% RSLogix 500 project I2P JOB 12 - ANDREW_HOEMMEN_BAK049.RSS, saved by version 10.00.00.00 %
PROJECT "ML03A"    % processor: Bul.1763 MicroLogix 1100 Series B %

PROGRAM FILES
  LAD 2   8 rungs

DATA FILES
  O0 OUTPUT  4 elements
  I1 INPUT  6 elements
  S2 STATUS  66 elements
  B3 BINARY  1 elements
  T4 TIMER  1 elements
  C5 COUNTER  1 elements
  R6 CONTROL  1 elements
  N7 INTEGER  1 elements
  F8 FLOAT  1 elements

LADDER 2
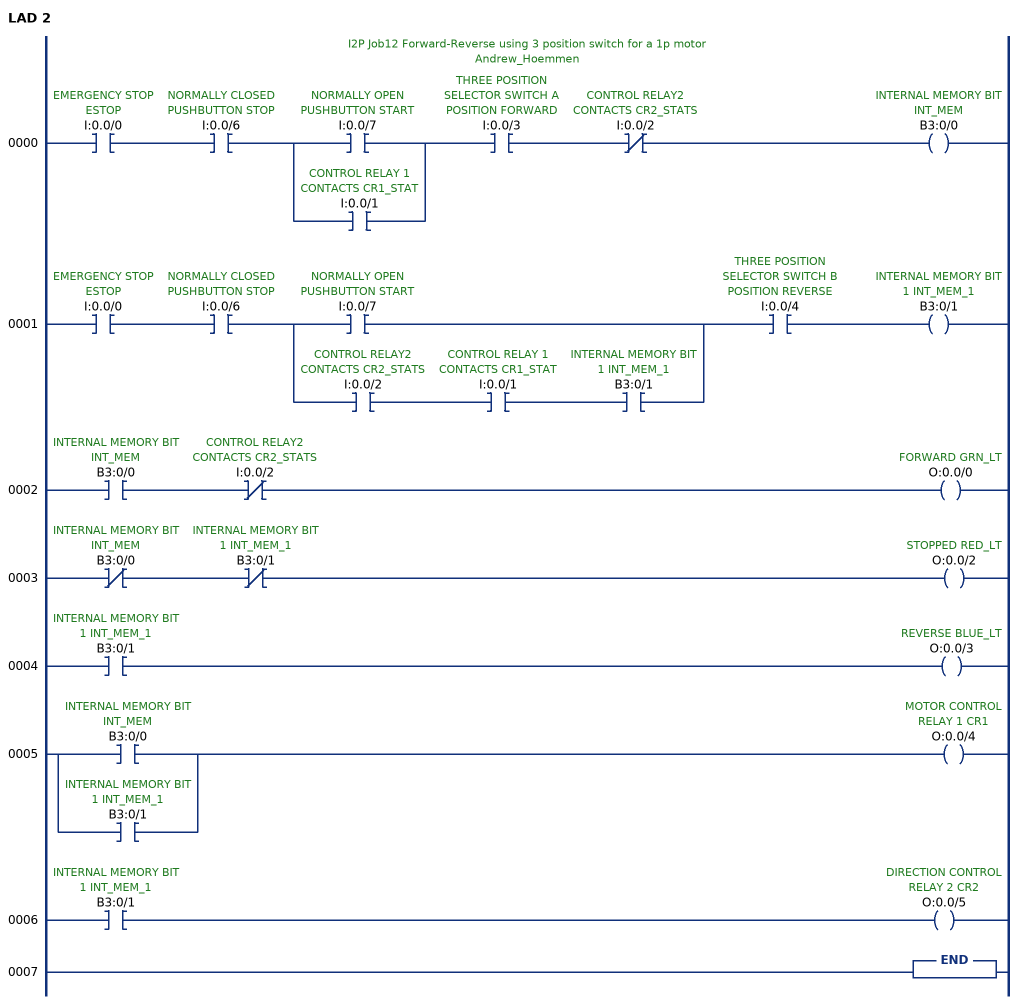
% Rung: 0 %
% I2P Job12 Forward-Reverse using 3 position switch for a 1p motor
% Andrew_Hoemmen %
SOR XIC I:0.0/0 XIC I:0.0/6 BST XIC I:0.0/7 NXB XIC I:0.0/1 BND XIC I:0.0/3 XIO I:0.0/2 OTE B3:0/0 EOR
%   I:0.0/0  ESTOP  "EMERGENCY STOP" %
%   I:0.0/6  STOP  "NORMALLY CLOSED PUSHBUTTON" %
%   I:0.0/7  START  "NORMALLY OPEN PUSHBUTTON" %
%   I:0.0/1  CR1_STAT  "CONTROL RELAY 1 CONTACTS" %
%   I:0.0/3  FORWARD  "THREE POSITION SELECTOR SWITCH A POSITION" %
%   I:0.0/2  CR2_STATS  "CONTROL RELAY2 CONTACTS" %
%   B3:0/0  INT_MEM  "INTERNAL MEMORY BIT" %
% Rung: 1 %
SOR XIC I:0.0/0 XIC I:0.0/6 BST XIC I:0.0/7 NXB XIC I:0.0/2 XIC I:0.0/1 XIC B3:0/1 BND XIC I:0.0/4 OTE B3:0/1 EOR
%   I:0.0/0  ESTOP  "EMERGENCY STOP" %
%   I:0.0/6  STOP  "NORMALLY CLOSED PUSHBUTTON" %
%   I:0.0/7  START  "NORMALLY OPEN PUSHBUTTON" %
%   I:0.0/2  CR2_STATS  "CONTROL RELAY2 CONTACTS" %
%   I:0.0/1  CR1_STAT  "CONTROL RELAY 1 CONTACTS" %
%   B3:0/1  INT_MEM_1  "INTERNAL MEMORY BIT 1" %
%   I:0.0/4  REVERSE  "THREE POSITION SELECTOR SWITCH B POSITION" %
% Rung: 2 %
SOR XIC B3:0/0 XIO I:0.0/2 OTE O:0.0/0 EOR
%   B3:0/0  INT_MEM  "INTERNAL MEMORY BIT" %
%   I:0.0/2  CR2_STATS  "CONTROL RELAY2 CONTACTS" %
%   O:0.0/0  GRN_LT  "FORWARD" %
% Rung: 3 %
SOR XIO B3:0/0 XIO B3:0/1 OTE O:0.0/2 EOR
%   B3:0/0  INT_MEM  "INTERNAL MEMORY BIT" %
%   B3:0/1  INT_MEM_1  "INTERNAL MEMORY BIT 1" %
%   O:0.0/2  RED_LT  "STOPPED" %
% Rung: 4 %
SOR XIC B3:0/1 OTE O:0.0/3 EOR
%   B3:0/1  INT_MEM_1  "INTERNAL MEMORY BIT 1" %
%   O:0.0/3  BLUE_LT  "REVERSE" %
% Rung: 5 %
SOR BST XIC B3:0/0 NXB XIC B3:0/1 BND OTE O:0.0/4 EOR
%   B3:0/0  INT_MEM  "INTERNAL MEMORY BIT" %
%   B3:0/1  INT_MEM_1  "INTERNAL MEMORY BIT 1" %
%   O:0.0/4  CR1  "MOTOR CONTROL RELAY 1" %
% Rung: 6 %
SOR XIC B3:0/1 OTE O:0.0/5 EOR
%   B3:0/1  INT_MEM_1  "INTERNAL MEMORY BIT 1" %
%   O:0.0/5  CR2  "DIRECTION CONTROL RELAY 2" %
% Rung: 7 %
SOR END EOR

OTHER DOCUMENTED ADDRESSES
  I:0.0/5  2PSS  "TWO POSITION SELECTOR SWITCH"
  I:0.0/8  PB3  "NORMALLY OPEN PUSHBUTTON"
  O:0.0/1  YEL_LT  "YELLOW LIGHT"
